FUNCTION Convert_DT_TO_LINT : Hresult
VAR_INPUT
	in : DT;
	out : REFERENCE TO LINT;
END_VAR
VAR
	converted : LINT;
END_VAR

converted := DT_TO_LINT(in);

IF (LINT_TO_DT(converted) <> in) THEN
	Convert_DT_TO_LINT := INCOMPATIBLE;
	RETURN;
END_IF

out := converted;

END_FUNCTION

(* stored: Version 1.1.0.1, ProductVersion 3.1.4024.12
   POU Convert_DT_TO_LINT: Id {c4e2af6f-f47a-4908-b066-c37458cb3cae}, SpecialFunc None *)
